PROGRAM MAIN
VAR
	testVar : INT :=0;
	
END_VAR

testVar := testVar + 1;

IF testVar > 100 THEN
	testVar := 0;
END_IF

END_PROGRAM

(* stored: Version 1.1.0.1, ProductVersion 3.1.4024.13
   POU MAIN: Id {bed3f892-980b-494c-a83f-03aad5f57fcb}, SpecialFunc None *)
